{attribute 'GeneratedUsingTerminal: EK1122-0000-0018'}
{attribute addProperty BoxType "EK1122-0000-0018"}
{attribute addProperty Id "Beckhoff_EP6xxxsub_EK1100EK1100_1FC0878B2A_0001_EP6001_0002_0020EP6001_40883D0360A_0002_EP6001_0002_0021EP6001_40883D0360A_0003_EP6002_0002_0016EP6002_2663B0AE108A_0004_EP6002_0002_0017EP6002_7F53816A108A_0005_EP6002_0002_0018EP6002_7F53816A108A_0006_EP6002_0002_0019EP6002_7F53816A108A_0007_EP6002_0002_0020EP6002_7F53816A108A_0008_EP6002_0002_0021EP6002_7F53816A108A_0009_EP6002_0002_0023EP6002_7BE6B617108A_0010_EP6002_0002_0024EP6002_7BE6B617108A_0011_EP6090_0000_0017EP6090_18BD01E922A_0012_EP6224_0002_0016EP6224_7D7C361B28A_0013_EP6224_0042_0016EP6224_77EE783032A_0014_EP6224_2022_0016EP6224_EDFF9F2F24A_0015_EP6224_2022_0017EP6224_EDFF9F2F24A_0016_EP6224_2022_0018EP6224_98EF241924A_0017_EP6224_3022_0016EP6224_EDFF9F2F24A_0018_EP6224_3022_0017EP6224_98EF241924A_0019_EP6228_0022_0016EP6228_FB34C73728A_0020_EP6228_0022_0017EP6228_FB34C73728A_0021_EP6228_0022_0018EP6228_FB34C73728A_0022_EP6228_0042_0016EP6228_495B58F436A_0023_EP6228_3032_0016EP6228_FB34C73728A_0024_EP6228_3132_0016EP6228_C205B54832A_0025_EP6228_3142_0016EP6228_C205B54832A_0026_EP6601_0002_0018EP6601_EEB2FEF410"}
{attribute addProperty CRC "1741432539"}
{attribute addProperty Size "1410"}
TYPE Beckhoff_EP6xxxEK1122_67CC26DB EXTENDS EK1122_1FC0878B :
STRUCT
	{attribute addProperty Name "Beckhoff EP6xxxsub EK1100"}
	{attribute addProperty PreviousPort "Beckhoff EP6xxxEK1122 : D"}
	Beckhoff_EP6xxxsub_EK1100 : EK1100_1FC0878B;
	{attribute addProperty Name "A_0001(EP6001-0002-0020)"}
	{attribute addProperty PreviousPort "Beckhoff EP6xxxsub EK1100 : C"}
	A_0001_EP6001_0002_0020 : EP6001_40883D03;
	{attribute addProperty Name "A_0002(EP6001-0002-0021)"}
	{attribute addProperty PreviousPort "A_0001(EP6001-0002-0020) : B"}
	A_0002_EP6001_0002_0021 : EP6001_40883D03;
	{attribute addProperty Name "A_0003(EP6002-0002-0016)"}
	{attribute addProperty PreviousPort "A_0002(EP6001-0002-0021) : B"}
	A_0003_EP6002_0002_0016 : EP6002_2663B0AE;
	{attribute addProperty Name "A_0004(EP6002-0002-0017)"}
	{attribute addProperty PreviousPort "A_0003(EP6002-0002-0016) : B"}
	A_0004_EP6002_0002_0017 : EP6002_7F53816A;
	{attribute addProperty Name "A_0005(EP6002-0002-0018)"}
	{attribute addProperty PreviousPort "A_0004(EP6002-0002-0017) : B"}
	A_0005_EP6002_0002_0018 : EP6002_7F53816A;
	{attribute addProperty Name "A_0006(EP6002-0002-0019)"}
	{attribute addProperty PreviousPort "A_0005(EP6002-0002-0018) : B"}
	A_0006_EP6002_0002_0019 : EP6002_7F53816A;
	{attribute addProperty Name "A_0007(EP6002-0002-0020)"}
	{attribute addProperty PreviousPort "A_0006(EP6002-0002-0019) : B"}
	A_0007_EP6002_0002_0020 : EP6002_7F53816A;
	{attribute addProperty Name "A_0008(EP6002-0002-0021)"}
	{attribute addProperty PreviousPort "A_0007(EP6002-0002-0020) : B"}
	A_0008_EP6002_0002_0021 : EP6002_7F53816A;
	{attribute addProperty Name "A_0009(EP6002-0002-0023)"}
	{attribute addProperty PreviousPort "A_0008(EP6002-0002-0021) : B"}
	A_0009_EP6002_0002_0023 : EP6002_7BE6B617;
	{attribute addProperty Name "A_0010(EP6002-0002-0024)"}
	{attribute addProperty PreviousPort "A_0009(EP6002-0002-0023) : B"}
	A_0010_EP6002_0002_0024 : EP6002_7BE6B617;
	{attribute addProperty Name "A_0011(EP6090-0000-0017)"}
	{attribute addProperty PreviousPort "A_0010(EP6002-0002-0024) : B"}
	A_0011_EP6090_0000_0017 : EP6090_18BD01E9;
	{attribute addProperty Name "A_0012(EP6224-0002-0016)"}
	{attribute addProperty PreviousPort "A_0011(EP6090-0000-0017) : B"}
	A_0012_EP6224_0002_0016 : EP6224_7D7C361B;
	{attribute addProperty Name "A_0013(EP6224-0042-0016)"}
	{attribute addProperty PreviousPort "A_0012(EP6224-0002-0016) : B"}
	A_0013_EP6224_0042_0016 : EP6224_77EE7830;
	{attribute addProperty Name "A_0014(EP6224-2022-0016)"}
	{attribute addProperty PreviousPort "A_0013(EP6224-0042-0016) : B"}
	A_0014_EP6224_2022_0016 : EP6224_EDFF9F2F;
	{attribute addProperty Name "A_0015(EP6224-2022-0017)"}
	{attribute addProperty PreviousPort "A_0014(EP6224-2022-0016) : B"}
	A_0015_EP6224_2022_0017 : EP6224_EDFF9F2F;
	{attribute addProperty Name "A_0016(EP6224-2022-0018)"}
	{attribute addProperty PreviousPort "A_0015(EP6224-2022-0017) : B"}
	A_0016_EP6224_2022_0018 : EP6224_98EF2419;
	{attribute addProperty Name "A_0017(EP6224-3022-0016)"}
	{attribute addProperty PreviousPort "A_0016(EP6224-2022-0018) : B"}
	A_0017_EP6224_3022_0016 : EP6224_EDFF9F2F;
	{attribute addProperty Name "A_0018(EP6224-3022-0017)"}
	{attribute addProperty PreviousPort "A_0017(EP6224-3022-0016) : B"}
	A_0018_EP6224_3022_0017 : EP6224_98EF2419;
	{attribute addProperty Name "A_0019(EP6228-0022-0016)"}
	{attribute addProperty PreviousPort "A_0018(EP6224-3022-0017) : B"}
	A_0019_EP6228_0022_0016 : EP6228_FB34C737;
	{attribute addProperty Name "A_0020(EP6228-0022-0017)"}
	{attribute addProperty PreviousPort "A_0019(EP6228-0022-0016) : B"}
	A_0020_EP6228_0022_0017 : EP6228_FB34C737;
	{attribute addProperty Name "A_0021(EP6228-0022-0018)"}
	{attribute addProperty PreviousPort "A_0020(EP6228-0022-0017) : B"}
	A_0021_EP6228_0022_0018 : EP6228_FB34C737;
	{attribute addProperty Name "A_0022(EP6228-0042-0016)"}
	{attribute addProperty PreviousPort "A_0021(EP6228-0022-0018) : B"}
	A_0022_EP6228_0042_0016 : EP6228_495B58F4;
	{attribute addProperty Name "A_0023(EP6228-3032-0016)"}
	{attribute addProperty PreviousPort "A_0022(EP6228-0042-0016) : B"}
	A_0023_EP6228_3032_0016 : EP6228_FB34C737;
	{attribute addProperty Name "A_0024(EP6228-3132-0016)"}
	{attribute addProperty PreviousPort "A_0023(EP6228-3032-0016) : B"}
	A_0024_EP6228_3132_0016 : EP6228_C205B548;
	{attribute addProperty Name "A_0025(EP6228-3142-0016)"}
	{attribute addProperty PreviousPort "A_0024(EP6228-3132-0016) : B"}
	A_0025_EP6228_3142_0016 : EP6228_C205B548;
	{attribute addProperty Name "A_0026(EP6601-0002-0018)"}
	{attribute addProperty PreviousPort "A_0025(EP6228-3142-0016) : B"}
	A_0026_EP6601_0002_0018 : EP6601_EEB2FEF4;
END_STRUCT
END_TYPE

(* stored: Version 1.2.0.0, ProductVersion 3.1.4024.11
   DUT Beckhoff_EP6xxxEK1122_67CC26DB: Id {152072ba-30c6-4f23-a580-f17af90b6908} *)
